TYPE MNG_APPLICATION_INPUTS_32BIT :
STRUCT
    NumSignals                     : INT     := 5         ;
    HallSensor1_00_IR : BOOL    := 0; (* ysics/Keksmodul/Keksmodul - relevant/HallSensor1?IR *)
    HallSensor2_00_IR : BOOL    := 0; (* ysics/Keksmodul/Keksmodul - relevant/HallSensor2?IR *)
    init_sensor_cookie_module_00_IR : BOOL    := 0; (* l/Keksmodul - relevant/init_sensor_cookie_module?IR *)
    kein_cookie_mehr_00_IR : BOOL    := 0; (* /Keksmodul/Keksmodul - relevant/kein_cookie_mehr?IR *)
    cookiebox_sensor_00_IR : BOOL    := 0; (* Physics://physics/Keksmodul/cookiebox_sensor?IR *)
END_STRUCT
END_TYPE

(* stored: Version 1.1.0.1, ProductVersion 3.1.0.25
   DUT MNG_APPLICATION_INPUTS_32BIT: Id {413e31a1-8a63-4a7e-b63f-9471650e1166} *)
